// TwinCAT 3 PLC project MotionSampleCode
// ProgramVersion: 3.1.4023.0
// libraries:
//   Tc2_Standard, * (Beckhoff Automation GmbH)
//   Tc2_System, * (Beckhoff Automation GmbH)
//   Tc3_Module, * (Beckhoff Automation GmbH)
// project tree:
//   RollerAxis/ EP7402_0xxx_Channel.TcPOU
//   RollerAxis/Structs/ DInputs.TcDUT, DOutputs.TcDUT, STMControl.TcDUT, STMInfoData.TcDUT, STMInputDevice.TcDUT, STMStatus.TcDUT, STMTargetVelocity.TcDUT
//   StepperAxis/ Ex70x7_DMC_Channel.TcPOU
//   StepperAxis/Structs/ StartType.TcDUT, StepperENCControl.TcDUT, StepperENCStatus.TcDUT, StepperPOSControl.TcDUT, StepperPOSStatus.TcDUT, StepperSTMControl.TcDUT, StepperSTMStatus.TcDUT
//   ServoAxis/ Exx72x1_DMC_Channel.TcPOU
//   ServoAxis/Structs/ DMC_Ins.TcDUT, DMC_Outs.TcDUT, DriveControl.TcDUT, DriveInputs.TcDUT, DriveOutputs.TcDUT, DriveStatus.TcDUT, PositioningControl.TcDUT, PositionStatus.TcDUT
//   / PlcTask.TcTTO
//   POUs/ MAIN.TcPOU
// real-time tasks:
//   TASK PlcTask: cycle T#10ms, priority 20, ADS port 350

CONFIGURATION MotionSampleCode
    RESOURCE PLC ON TwinCAT3
        TASK PlcTask(INTERVAL := T#10ms, PRIORITY := 20);
        PROGRAM MAIN WITH PlcTask : MAIN;
    END_RESOURCE
END_CONFIGURATION

// ---- RollerAxis/Structs/DInputs.TcDUT
TYPE DInputs :
STRUCT
	input1 : BOOL;
	input2 : BOOL;
	input3 : BOOL;
	input4 : BOOL;
	controlInput1 : BOOL;
	controlInput2 : BOOL;
	controlInput3 : BOOL;
	controlInput4 : BOOL;
END_STRUCT
END_TYPE

// ---- RollerAxis/Structs/DOutputs.TcDUT
TYPE DOutputs :
STRUCT
	output1 : BOOL;
	output2 : BOOL;
	output3 : BOOL;
	output4 : BOOL;
	controlOutput1 : BOOL;
	controlOutput2 : BOOL;
	controlOutput3 : BOOL;
	controlOutput4 : BOOL;
END_STRUCT
END_TYPE

// ---- RollerAxis/Structs/STMControl.TcDUT
TYPE STMControl :
STRUCT
	enable : BOOL;
	reset : BOOL;
	invertDirection : BOOL;
	brakeOutput : BOOL;
END_STRUCT
END_TYPE

// ---- RollerAxis/Structs/STMInfoData.TcDUT
TYPE STMInfoData :
STRUCT
	infoData1 : UINT;
	infoData2 : UINT;
	infoData3 : UINT;
END_STRUCT
END_TYPE

// ---- RollerAxis/Structs/STMInputDevice.TcDUT
TYPE STMInputDevice :
STRUCT
	deviceUnderVoltage : BOOL;
	deviceOverVoltage : BOOL;
	overTemperatureWarning : BOOL;
	overTemperatureError : BOOL;
	generalHWError : BOOL;
	chn1OpenLoad : BOOL;
	chn1ShortCircuit : BOOL;
	chn1MotorOverloadI2TWarning : BOOL;
	chn1MotorOverloadI2TError : BOOL;
	chn1AmplifierOverloadI2TWarning : BOOL;
	chn1AmplifierOverloadI2TError : BOOL;
	chn1InLimit : BOOL;
	chn1CommutationError : BOOL;
	chn2OpenLoad : BOOL;
	chn2ShortCircuit : BOOL;
	chn2MotorOverloadI2TWarning : BOOL;
	chn2MotorOverloadI2TError : BOOL;
	chn2AmplifierOverloadI2TWarning : BOOL;
	chn2AmplifierOverloadI2TError : BOOL;
	chn2InLimit : BOOL;
	chn2CommutationError : BOOL;
END_STRUCT
END_TYPE

// ---- RollerAxis/Structs/STMStatus.TcDUT
TYPE STMStatus :
STRUCT
	readyToEnable : BOOL;
	ready : BOOL;
	warning : BOOL;
	error : BOOL;
	movingPositive : BOOL;
	movingNegative : BOOL;
	txPDOToggle : BOOL;
END_STRUCT
END_TYPE

// ---- RollerAxis/Structs/STMTargetVelocity.TcDUT
TYPE STMTargetVelocity :
STRUCT
	velocity : INT;
	acceleration : UINT;
	deceleration : UINT;
END_STRUCT
END_TYPE

// ---- StepperAxis/Structs/StartType.TcDUT
{attribute 'qualified_only'}
{attribute 'strict'}
TYPE StartType :
(
	Absolute := 1,
	Relative := 2,
	VeloPositive := 3,
	VeloNegative := 4,
	Calibrate := 24576 
);
END_TYPE

// ---- StepperAxis/Structs/StepperENCControl.TcDUT
TYPE StepperENCControl :
STRUCT
	EnableLatchC : BOOL;
	EnableLatchPositiveEdge : BOOL;
	SetCounter : BOOL;
	EnableLatchNegativeEdge : BOOL;
	SetCounterValue : UDINT;
END_STRUCT
END_TYPE

// ---- StepperAxis/Structs/StepperENCStatus.TcDUT
TYPE StepperENCStatus :
STRUCT
	LatchCValid : BOOL;
	LatchExternalValid : BOOL;
	SetCounterDone : BOOL;
	CounterUnderflow : BOOL;
	CounterOverflow : BOOL;
	ExtrapolationStall : BOOL;
	StatusInputA : BOOL;
	StatusInputB : BOOL;
	StatusInputC : BOOL;
	StatusExternLatch : BOOL;
	SyncError : BOOL;
	TxPDOToggle : BOOL;
	CounterValue : UDINT;
	LatchValue : UDINT;
END_STRUCT
END_TYPE

// ---- StepperAxis/Structs/StepperPOSControl.TcDUT
TYPE StepperPOSControl :
STRUCT
	Execute : BOOL;
	EmergencyStop : BOOL;
	TargetPosition : UDINT;
	Velocity : INT;
	StartType : UINT;
	Acceleration : UINT;
	Deceleration : UINT;
END_STRUCT
END_TYPE

// ---- StepperAxis/Structs/StepperPOSStatus.TcDUT
TYPE StepperPOSStatus :
STRUCT
	Busy : BOOL;
	InTarget : BOOL;
	Warning : BOOL;
	Error : BOOL;
	Calibrated : BOOL;
	Accelerate : BOOL;
	Decelerate : BOOL;
	ReadyToExecute : BOOL;
	ActualPosition : UDINT;
	ActualVelocity : INT;
	ActualDriveTime : UDINT;
END_STRUCT
END_TYPE

// ---- StepperAxis/Structs/StepperSTMControl.TcDUT
TYPE StepperSTMControl :
STRUCT
	Enable : BOOL;
	Reset : BOOL;
	ReduceTorque : BOOL;
	DigitalOutput1 : BOOL;
END_STRUCT
END_TYPE

// ---- StepperAxis/Structs/StepperSTMStatus.TcDUT
TYPE StepperSTMStatus :
STRUCT
	ReadyToEnable : BOOL;
	Ready : BOOL;
	Warning : BOOL;
	Error : BOOL;
	MovingPositive : BOOL;
	MovingNegative : BOOL;
	MotorStall : BOOL;
	DigitalInput1 : BOOL;
	DigitalInput2 : BOOL;
	SyncError : BOOL;
	TxPDOToggle : BOOL;
END_STRUCT
END_TYPE

// ---- ServoAxis/Structs/DMC_Ins.TcDUT
TYPE DMC_Ins :
STRUCT
	DMC_Inputs : DriveInputs;
	DMC_POS_Status : PositionStatus;
	DMC_Drv_Status : DriveStatus;
END_STRUCT
END_TYPE

// ---- ServoAxis/Structs/DMC_Outs.TcDUT
TYPE DMC_Outs :
STRUCT
	DMC_DrvOuts : DriveOutputs;
	DMC_Drv_Ctrl : DriveControl;
	DMC_POS_Ctrl : PositioningControl;
END_STRUCT
END_TYPE

// ---- ServoAxis/Structs/DriveControl.TcDUT
TYPE DriveControl :
STRUCT
	Enable : BOOL;
	Reset : BOOL;
END_STRUCT
END_TYPE

// ---- ServoAxis/Structs/DriveInputs.TcDUT
TYPE DriveInputs :
STRUCT
	SetPosition : UDINT;
	SetVelocity : INT;
	ActualDriveTime : UDINT;
	ActualPositionLag : DINT;
	ActualVelocity : INT;
	ActualPosition : UDINT;
	ErrorId : UDINT;
	InputCycleCounter : USINT;
	LatchValue : UDINT;
	CyclicInfoData1 : INT;
	CyclicInforData2 : INT;
END_STRUCT
END_TYPE

// ---- ServoAxis/Structs/DriveOutputs.TcDUT
TYPE DriveOutputs :
STRUCT
	SetCounterValue : UDINT;
	TargetPosition : UDINT;
	TargetVelocity : INT;
	StartType : UINT;
	TargetAcceleration : UINT;
	TargetDeceleration : UINT;
END_STRUCT
END_TYPE

// ---- ServoAxis/Structs/DriveStatus.TcDUT
TYPE DriveStatus :
STRUCT
	ReadyToEnable : BOOL;
	Ready : BOOL;
	Warning : BOOL;
	Error : BOOL;
	MovingPositive : BOOL;
	MovingNegative : BOOL;
	DigitalInput1 : BOOL;
	DigitalInput2 : BOOL;
END_STRUCT
END_TYPE

// ---- ServoAxis/Structs/PositioningControl.TcDUT
TYPE PositioningControl :
STRUCT
	Execute : BOOL;
	EmergencyStop : BOOL;
END_STRUCT
END_TYPE

// ---- ServoAxis/Structs/PositionStatus.TcDUT
TYPE PositionStatus :
STRUCT
	Busy : BOOL;
	InTarget : BOOL;
	Warning : BOOL;
	Error : BOOL;
	Calibrated : BOOL;
	Accelerate : BOOL;
	Decelerate : BOOL;
	ReadyToExecute : BOOL;
END_STRUCT
END_TYPE

// ---- POUs/MAIN.TcPOU
PROGRAM MAIN
VAR
END_VAR

END_PROGRAM

// ---- RollerAxis/EP7402_0xxx_Channel.TcPOU
FUNCTION_BLOCK EP7402_0xxx_Channel
VAR_INPUT
END_VAR
VAR_OUTPUT
END_VAR
VAR
	DI_Inputs AT%I* : DInputs;
	DO_Outputs AT%Q* : DOutputs;
	STM_Control AT%Q* : STMControl;
	STM_Info_data AT%I* : STMInfoData;
	STM_Input_Device AT%I* : STMInputDevice;
	STM_Status AT%I* : STMStatus;
	STM_Target_Velocity AT%Q* : STMTargetVelocity;
	
	_acceleration : UINT := 100;
	_deceleration : UINT := 100;
	
	State :(
		_00_mWait,
        _01_mReset,
        _02_mEnable,
		_03_mStop,
		_04_RunAtVelo,
		_05_mDisable);
		
	tonHoldHigh	: ton;
		
END_VAR

CASE State OF
        _00_mWait : 
			;
        _01_mReset : 
			STM_Control.reset := TRUE;
			tonHoldHigh(in := TRUE, pt := T#500MS);
			IF tonHoldHigh.Q THEN
				STM_Control.reset := FALSE;
				IF STM_Status.error = FALSE AND
					STM_Status.warning = FALSE AND
					STM_Status.ready = TRUE
				THEN
					State := _00_mWait;
					tonHoldHigh(in := FALSE);
				END_IF
			END_IF
			
        _02_mEnable : 
			IF STM_Status.error THEN				
				State := _01_mReset;
			ELSE
				STM_Control.enable := TRUE;			
			END_IF

			
		_04_RunAtVelo :
			;
			
		_03_mStop : 
			STM_Target_Velocity.velocity := 0;
			IF STM_Status.ready THEN	
				State := _02_mEnable;
			END_IF
			
		_05_mDisable:
			STM_Control.enable := FALSE;
			State := _00_mWait;
		
			
END_CASE

PROPERTY PUBLIC Acceleration : uint
GET
Acceleration := _acceleration;
END_GET
SET
_acceleration := Acceleration;
END_SET
END_PROPERTY

PROPERTY PUBLIC Deceleration : uint
GET
Deceleration := _deceleration;
END_GET
SET
_deceleration := Deceleration;
END_SET
END_PROPERTY

METHOD Disable : BOOL
VAR_INPUT
END_VAR
IF STM_Status.ready THEN
	State := _05_mDisable;
END_IF
END_METHOD

METHOD Enable : BOOL
VAR_INPUT
END_VAR
IF STM_Status.readyToEnable THEN
	State := _02_mEnable;
END_IF
END_METHOD

METHOD MoveNeg : BOOL
VAR_INPUT
END_VAR
STM_Control.invertDirection := TRUE;
STM_Target_Velocity.velocity := 6000;
STM_Target_Velocity.acceleration := _acceleration;
STM_Target_Velocity.deceleration := _deceleration;
State := _04_RunAtVelo;
END_METHOD

METHOD MovePos : BOOL
VAR_INPUT
END_VAR
STM_Control.invertDirection := FALSE;
STM_Target_Velocity.velocity := 6000;
STM_Target_Velocity.acceleration := _acceleration;
STM_Target_Velocity.deceleration := _deceleration;
State := _04_RunAtVelo;
END_METHOD

METHOD Reset : BOOL
VAR_INPUT
END_VAR
IF STM_Status.error OR STM_Status.warning THEN
	State := _01_mReset;
END_IF
END_METHOD

METHOD Stop : BOOL
VAR_INPUT
END_VAR
IF STM_Status.movingNegative OR STM_Status.movingPositive THEN
	State := _03_mStop;
END_IF
END_METHOD

END_FUNCTION_BLOCK

// ---- StepperAxis/Ex70x7_DMC_Channel.TcPOU
FUNCTION_BLOCK Ex70x7_DMC_Channel
VAR_INPUT
END_VAR
VAR_OUTPUT
END_VAR
VAR
	ENCStatus AT%I* : StepperENCStatus;
	STMStatus AT%I* : StepperSTMStatus;
	POSStatus AT%I* : StepperPOSStatus;
	
	ENCControl AT%Q* : StepperENCControl;
	STMControl AT%Q* : StepperSTMControl;
	POSControl AT%Q* : StepperPOSControl;
	
	_InTarget : BOOL;
	
	State :(
		_00_mWait,
        _01_mReset,
        _02_mEnable,
		_06_mGotoPosition,
		_07_mStop,
		_08_mSetPosition,
		_09_RunAtExternalVelo,
		_10_Disable);
		
	tonHoldHigh				: ton;
END_VAR

CASE State OF
        _00_mWait : 
			;
        _01_mReset : 
			STMControl.Reset := TRUE;
			tonHoldHigh(in := TRUE, pt := T#500MS);
			IF tonHoldHigh.Q THEN
				STMControl.Reset := FALSE;
				IF STMStatus.Error = FALSE AND
					STMStatus.Warning = FALSE AND
					STMStatus.Ready = TRUE
				THEN
					State := _00_mWait;
					tonHoldHigh(in := FALSE, pt := T#500MS);
				END_IF
			END_IF
			
        _02_mEnable : 
			IF STMStatus.Error THEN				
				State := _01_mReset;
			ELSE
				STMControl.Enable := TRUE;			
			END_IF
			
		_06_mGotoPosition :
			POSControl.Execute := TRUE;
			_InTarget := FALSE;
			IF POSStatus.InTarget THEN
				State := _02_mEnable;
				POSControl.Execute := FALSE;
				_InTarget := TRUE;
			END_IF
			
		_07_mStop : 
			POSControl.Execute := FALSE;
			IF POSStatus.ReadyToExecute THEN	
				State := _02_mEnable;
			END_IF
			
		_08_mSetPosition :
			POSControl.Execute := TRUE;
			
			IF POSStatus.Calibrated THEN
				POSControl.Execute := FALSE;
				State := _02_mEnable;
			END_IF
			
		_09_RunAtExternalVelo :
			POSControl.Execute := TRUE;
			_InTarget := false;
			
		_10_Disable:
			STMControl.Enable := FALSE;
			State := _00_mWait;
		
			
END_CASE

PROPERTY ActualPosition : lreal
GET
ActualPosition := UDINT_TO_LREAL( POSStatus.ActualPosition)/8062.72;
END_GET
END_PROPERTY

PROPERTY ActualVelocity : int
GET
ActualVelocity := POSStatus.ActualVelocity;
END_GET
END_PROPERTY

METHOD CalibrateMotor : BOOL
VAR_INPUT
END_VAR
IF State = _02_mEnable THEN
	State := _08_mSetPosition;
	//POSControl.Velocity := REAL_TO_INT( Velocity*252);
	POSControl.StartType := StartType.Calibrate;
	//POSControl.TargetPosition := LREAL_TO_UDINT(Position*8062.72);
	//POSControl.TargetPosition := LREAL_TO_UDINT(Position*10);
END_IF
END_METHOD

METHOD Disable : BOOL
VAR_INPUT
END_VAR
IF STMStatus.Ready THEN
	State := _10_Disable;
END_IF
END_METHOD

METHOD Enable : BOOL
VAR_INPUT
END_VAR
IF STMStatus.ReadyToEnable THEN
	State := _02_mEnable;
END_IF
END_METHOD

METHOD GoToPosition : BOOL
VAR_INPUT
	Position : LREAL;
	Velocity : REAL;
END_VAR
IF State = _02_mEnable THEN
	State := _06_mGoToPosition;
	POSControl.Velocity := REAL_TO_INT( Velocity*252);
	POSControl.StartType := StartType.Absolute;
	POSControl.TargetPosition := LREAL_TO_UDINT(Position*8062.72);
END_IF
END_METHOD

PROPERTY InTarget : bool
GET
InTarget := _InTarget;
END_GET
END_PROPERTY

METHOD MoveAtVelocity : BOOL
VAR_INPUT
	Velocity : REAL;
END_VAR
IF State = _02_mEnable THEN
	State := _09_RunAtExternalVelo;
	POSControl.Velocity := REAL_TO_INT( Velocity*252);
	POSControl.StartType := StartType.VeloPositive;
END_IF
END_METHOD

PROPERTY Ready : bool
GET
Ready := STMStatus.Ready;
END_GET
END_PROPERTY

METHOD Reset : BOOL
VAR_INPUT
END_VAR
IF STMStatus.Error OR STMStatus.Warning OR POSStatus.Error THEN
	State := _01_mReset;
END_IF
END_METHOD

METHOD Stop : BOOL
VAR_INPUT
END_VAR
IF POSControl.Execute THEN
	State  := _07_mStop;
END_IF
END_METHOD

END_FUNCTION_BLOCK

// ---- ServoAxis/Exx72x1_DMC_Channel.TcPOU
FUNCTION_BLOCK Exx72x1_DMC_Channel
VAR_INPUT
END_VAR
VAR_OUTPUT
END_VAR
VAR
	//Properties
	_acceleration : UINT := 4000; 	//default to 4s accel
	_deceleration : UINT := 4000;	//default to 4s decel
	_startType : UINT := 1; 		//default to abs moves
	_scale : REAL := 360; 			//default to 360 degree scale factor
	
	//Locals
	dmc_inputs AT%I* : DMC_Ins;
	dmc_outputs AT%q* : DMC_Outs;
	xMove: BOOL;
	iMove: INT;
	
	posDemand : REAL;
	currentPos : REAL;
END_VAR

MoveSequence();

dmc_outputs.DMC_DrvOuts.TargetPosition := REAL_TO_UDINT(posDemand * (1048576/360));
currentPos := UDINT_TO_REAL( dmc_inputs.DMC_Inputs.ActualPosition)*(360.0/1048576.0);

PROPERTY PUBLIC Acceleration : uint
GET
Acceleration := _acceleration;
END_GET
SET
_acceleration := Acceleration;
END_SET
END_PROPERTY

PROPERTY PUBLIC Deceleration : uint
GET
Deceleration := _deceleration;
END_GET
SET
_deceleration := Deceleration;
END_SET
END_PROPERTY

METHOD PUBLIC Enable : BOOL
VAR_INPUT
END_VAR
IF dmc_inputs.DMC_Drv_Status.ReadyToEnable THEN
	dmc_outputs.DMC_Drv_Ctrl.Enable := TRUE;
END_IF
END_METHOD

PROPERTY PUBLIC Enabled : bool
GET
Enabled := dmc_inputs.DMC_Drv_Status.Ready AND dmc_inputs.DMC_POS_Status.ReadyToExecute;
END_GET
END_PROPERTY

PROPERTY PUBLIC Error : bool
GET
Error := dmc_inputs.DMC_Drv_Status.Error;
END_GET
END_PROPERTY

METHOD PUBLIC MoveAxis : BOOL
VAR_INPUT
	PositioningControl : real;
	Velocity : INT;
END_VAR
dmc_outputs.DMC_DrvOuts.TargetPosition := REAL_TO_UDINT(PositioningControl*(1048576/_scale));
dmc_outputs.DMC_DrvOuts.TargetVelocity := Velocity;
dmc_outputs.DMC_DrvOuts.StartType := _startType;
dmc_outputs.DMC_DrvOuts.TargetAcceleration := _acceleration;
dmc_outputs.DMC_DrvOuts.TargetDeceleration := _deceleration;
xMove := TRUE;
MoveAxis := TRUE;
END_METHOD

METHOD PRIVATE MoveSequence : BOOL
VAR_INPUT
END_VAR
CASE iMove OF 
	0: 
		IF dmc_inputs.DMC_POS_Status.ReadyToExecute AND xMove THEN
			xMove := FALSE;
			iMove := 10;
		END_IF
	10:
		dmc_outputs.DMC_POS_Ctrl.Execute := TRUE;
		IF dmc_inputs.DMC_POS_Status.Busy THEN
			iMove := 20;
		END_IF
	20:
		IF NOT dmc_inputs.DMC_POS_Status.Busy THEN
			IF dmc_inputs.DMC_POS_Status.InTarget THEN
				iMove := 0;
			ELSE
				iMove :=99;
			END_IF
			dmc_outputs.DMC_POS_Ctrl.Execute := FALSE;
		END_IF
END_CASE
END_METHOD

PROPERTY PUBLIC Scale : real
GET
Scale := _scale;
END_GET
SET
_scale := Scale;
END_SET
END_PROPERTY

PROPERTY PUBLIC StartType : uint
GET
StartType := _startType;
END_GET
SET
_startType := StartType;
END_SET
END_PROPERTY

END_FUNCTION_BLOCK
